{attribute 'linkalways'} 
{attribute 'no_explicit_call' := 'This FB is a CLASS and must be accessed using methods or properties'}
{attribute 'enable_dynamic_creation'}
FUNCTION_BLOCK _ETcVnDistanceTransformationMask EXTENDS EnumDatatypeBase
VAR
	localData : ETcVnDistanceTransformationMask;
	activeData : REFERENCE TO ETcVnDistanceTransformationMask;
	enumBaseDatatype : _DINT(localData);
END_VAR

METHOD PRIVATE AddLocalEnumeration
VAR_INPUT
	Enumeration : T_MAXSTRING;
	Value : ETcVnDistanceTransformationMask;
END_VAR
AddEnumeration(Enumeration, Value);
END_METHOD

PROPERTY PUBLIC Address : PVOID
GET
Address := ADR(activeData);
END_GET
END_PROPERTY

METHOD PUBLIC ClearReference
VAR_INPUT
END_VAR
activeData REF= localData;
SetBaseDatatypeReference();
END_METHOD

METHOD PUBLIC Clone : I_Datatype
VAR
    pClone : POINTER TO _ETcVnDistanceTransformationMask;
END_VAR
pClone := __NEW(_ETcVnDistanceTransformationMask(InitialValue := Value));
Clone := pClone^;
END_METHOD

METHOD FB_init : BOOL
VAR_INPUT
	bInitRetains : BOOL; // if TRUE, the retain variables are initialized (warm start / cold start)
	bInCopyCode : BOOL;  // if TRUE, the instance afterwards gets moved into the copy code (online change)
	InitialValue : ETcVnDistanceTransformationMask;
END_VAR
localData := InitialValue;
AddBaseDatatype(enumBaseDatatype);
ClearReference();

AddLocalEnumeration('TCVN_DTM_PRECISE', ETcVnDistanceTransformationMask.TCVN_DTM_PRECISE);
AddLocalEnumeration('TCVN_DTM_3', ETcVnDistanceTransformationMask.TCVN_DTM_3);
AddLocalEnumeration('TCVN_DTM_5', ETcVnDistanceTransformationMask.TCVN_DTM_5);
END_METHOD

PROPERTY PUBLIC Identifier : T_MAXSTRING
GET
Identifier := 'ETcVnDistanceTransformationMask';
END_GET
END_PROPERTY

METHOD IsEnumeratorValueEqual : BOOL
VAR_INPUT
	Enumerator : I_KeyValueForwardEnumerator;
END_VAR
VAR
	storedValue : ETcVnDistanceTransformationMask;
END_VAR
IF NOT Enumerator.TryGet(storedValue) THEN
	RETURN;
END_IF

IsEnumeratorValueEqual := storedValue = activeData;
END_METHOD

METHOD PUBLIC MakeReferenceTo
VAR_INPUT
	ReferenceTarget : REFERENCE TO ETcVnDistanceTransformationMask;
END_VAR
activeData REF= ReferenceTarget;
SetBaseDatatypeReference();
END_METHOD

METHOD PROTECTED SetBaseDatatypeReference
VAR_INPUT
END_VAR
enumBaseDatatype.MakeReferenceTo(activeData);
END_METHOD

PROPERTY PUBLIC Size : UDINT
GET
Size := SIZEOF(activeData);
END_GET
END_PROPERTY

METHOD TryMakeReferenceTo : BOOL
VAR_INPUT
	Target : I_Datatype;
END_VAR
VAR
	targetAsEnum : I_EnumDatatype;
	pTargetData : POINTER TO ETcVnDistanceTransformationMask;
END_VAR
IF NOT Target.TryResolveAsEnumDatatype(targetAsEnum) THEN
	RETURN;
END_IF

IF targetAsEnum.Identifier <> Identifier THEN
	RETURN;
END_IF

pTargetData := Target.Address;
activeData REF= pTargetData^;
SetBaseDatatypeReference();
TryMakeReferenceTo := TRUE;
END_METHOD

PROPERTY PUBLIC Value : ETcVnDistanceTransformationMask
GET
Value := activeData;
END_GET
SET
activeData := Value;
END_SET
END_PROPERTY

END_FUNCTION_BLOCK

(* stored: Version 1.1.0.1
   POU _ETcVnDistanceTransformationMask: Id {f7ef2f2a-1891-47e6-ace7-e1a8016cb18d}, SpecialFunc None
   Folder Constructor: Id {730253d8-93a2-4633-8c40-9b1ac68ceed5}
   Folder Private: Id {2b7cf6a7-8ba0-42b0-97bf-9c47e8703b95}
   Folder Protected: Id {1a0c6afc-9db6-4cb7-bfb0-7fa4b27116c9}
   Method AddLocalEnumeration: Id {68e23d6f-b017-4f6f-9256-ada88cff4ff5}
   Property Address: Id {f3680436-887d-43a2-b3f4-ffc07fdd8a9a}
   Get Get: Id {e03059ef-1365-44b5-a92c-fe889ac4e243}
   Method ClearReference: Id {ad90983d-734c-4eb1-a67b-435ff3501292}
   Method Clone: Id {1bb0f1dd-ff72-4ede-ada0-9475f1bada88}
   Method FB_init: Id {0dc2931c-9100-4f33-ade5-bef9ad3eadb5}
   Property Identifier: Id {de81f1b5-d127-4ae8-9d0d-e385048bf18d}
   Get Get: Id {96f35df6-a4d9-43fb-9464-dccdc9d3be28}
   Method IsEnumeratorValueEqual: Id {f180e012-8dfd-4440-8806-5974f0bc3fa1}
   Method MakeReferenceTo: Id {273a8522-57c6-48b4-86a9-41561db086f4}
   Method SetBaseDatatypeReference: Id {56587564-a93c-4f77-abb3-deadc029786f}
   Property Size: Id {c3ee0e6e-215b-4acd-a059-0ea50c1bdaec}
   Get Get: Id {65083c1e-9b47-45b9-a9ad-9429976e5535}
   Method TryMakeReferenceTo: Id {fc7c1fe7-602d-4026-bc4f-7fcd33cf816e}
   Property Value: Id {ab2a0f32-24bc-4eda-b592-651ad29ce569}
   Get Get: Id {a62e4d79-cdf6-4cfc-bfce-6f2879583169}
   Set Set: Id {01b2ec90-02c0-4be2-9eac-bc67cf3b9893} *)
